// Mitsubishi GX Works2 project: PLC_GROUP7   PLC: FX3G

// global labels: Global1
VAR_GLOBAL
  Switch_Workday AT X007 : BOOL;
  Switch_Cream AT X011 : BOOL;
  Light_Workday AT Y007 : BOOL;
  Light_Transporting0 AT Y000 : BOOL;
  Light_Transporting1 AT Y001 : BOOL;
  Switch_Sample AT X006 : BOOL;
  Light_Chocolate AT Y003 : BOOL;
  Wrap_Krembo AT X000 : BOOL;
  Light_5Krembos AT Y002 : BOOL;
  Stock_Cream AT D1100 : REAL;
  Stock_Chocolate AT D1102 : REAL;
  Stock_Biscuits AT D1104 : REAL;
END_VAR
VAR_GLOBAL CONSTANT
  Serving_Cream : REAL := 300;
  Serving_Chocolate_Normal : REAL := 120;
  Serving_Biscuits : REAL := 6;
  Starting_Cream : REAL := 900;
  Starting_Chocolate : REAL := 500;
  Starting_Biscuits : REAL := 30;
END_VAR
VAR_GLOBAL
  Container_Cream AT D1114 : REAL;
  Container_Chocolate AT D1116 : REAL;
END_VAR
VAR_GLOBAL CONSTANT
  Serving_Chocolate_Double : REAL := 240;
END_VAR
VAR_GLOBAL
  Switch_MachineA AT X010 : BOOL;
  MachineA_on AT M0 : BOOL;
  MachineA_Stop AT X005 : BOOL;
  Sens_30 AT X002 : BOOL;
  Sens_15 AT X001 : BOOL;
  Light_MachineA_Work AT Y004 : BOOL;
  Sens_camera AT X003 : BOOL;
  Light_alternate AT M1 : BOOL;
  Timer_alternate AT TC1 : BOOL;
END_VAR
VAR_GLOBAL CONSTANT
  Timer_alternate_duration : INT := 40;
END_VAR
VAR_GLOBAL
  Timer_alterante_State AT TS1 : BOOL;
  Light_state AT M2 : BOOL;
  Light_Y0_Timer AT TC2 : BOOL;
  Light_Y1_Timer AT TC3 : BOOL;
  Light_Y0_State AT TS2 : BOOL;
  Light_Y1_State AT TS3 : BOOL;
END_VAR
VAR_GLOBAL CONSTANT
  Timer_Alternate_Switch : INT := 5;
END_VAR
VAR_GLOBAL
  Analog_Input1 AT D8280 : INT;
END_VAR
VAR_GLOBAL CONSTANT
  Chocolate_Coat : INT := 5;
  Div_400 : INT := 400;
END_VAR
VAR_GLOBAL
  Dipping_Timer AT TC4 : BOOL;
  Dipping_State AT TS4 : BOOL;
END_VAR
VAR_GLOBAL CONSTANT
  Dipping_Duration : INT := 50;
END_VAR
VAR_GLOBAL
  krembo_dipping AT M3 : BOOL;
END_VAR
VAR_GLOBAL CONSTANT
  krembo_5Limit : INT := 5;
END_VAR
VAR_GLOBAL
  krembo_5Count AT CC1 : BOOL;
  krembo_State AT CS1 : BOOL;
  Counter_5Krembo AT CN1 : INT;
END_VAR
VAR_GLOBAL CONSTANT
  Krembo_6Limit : INT := 6;
END_VAR
VAR_GLOBAL
  Krembo_Second_State AT CS2 : BOOL;
  Counter_6Krembo AT CN2 : INT;
  Krembo_6Count AT CC2 : BOOL;
  Light_Y2_Help AT M5 : BOOL;
  Total_Krembo AT D1118 : REAL;
  Analog_Output AT D8282 : INT;
  Light_Alternate2 AT M4 : BOOL;
  Light_alternate_endDay AT M6 : BOOL;
  Timer_endDay AT TC5 : BOOL;
  Timer_endDay_State AT TS5 : BOOL;
END_VAR
VAR_GLOBAL CONSTANT
  EndDay_Duration : INT := 30;
END_VAR
VAR_GLOBAL
  Light_alternate_endDay2 AT M7 : BOOL;
  Timer_endDay2 AT TC6 : BOOL;
  Timer_endDay_State2 AT TS6 : BOOL;
  Got_Biscuits AT M11 : BOOL;
  Got_Cream AT M12 : BOOL;
  Got_Chocolate AT M13 : BOOL;
  Timer_endDay3 AT TC7 : BOOL;
  Timer_endDay_State3 AT TS7 : BOOL;
  End_Blink_Light2 AT M14 : BOOL;
  Sens_Pack AT X004 : BOOL;
  End_Blink_Light AT M16 : BOOL;
  End_Iteration AT M17 : BOOL;
  Fictive_Light_Workday AT M18 : BOOL;
END_VAR
VAR_GLOBAL CONSTANT
  Mul_40 : INT := 40;
END_VAR

// task Task_01 (event TRUE, interval 0, priority 31): POU_01

PROGRAM POU_01
(* structured ladder/FBD written out as ST: instructions are called as NAME(EN, inputs, outputs); _pN, _eN, _tN stand for wires *)
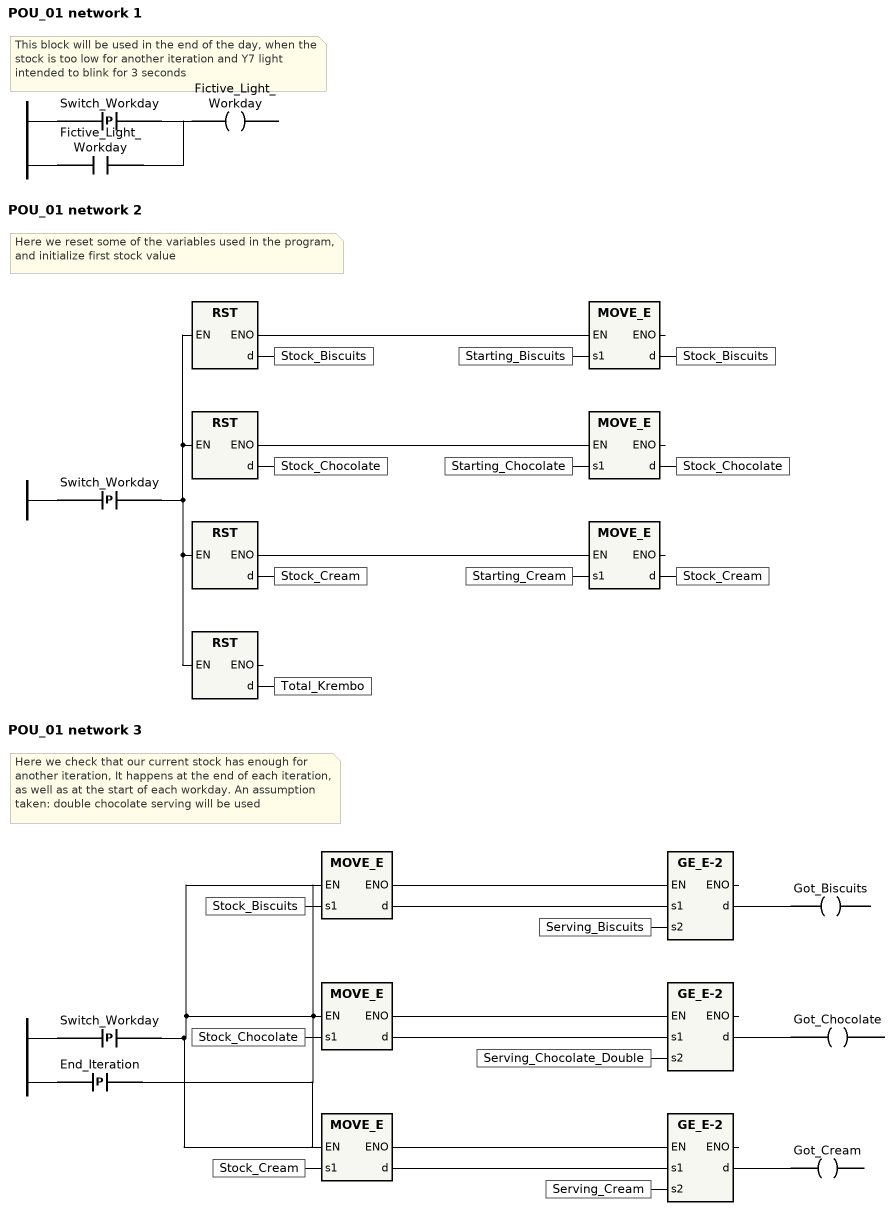
(* network 1 *)
(* This block will be used in the end of the day, when the stock is too low for another iteration and Y7 light intended to blink for 3 seconds *)
Fictive_Light_Workday := LDP(TRUE, Switch_Workday) OR Fictive_Light_Workday;
(* network 2 *)
(* Here we reset some of the variables used in the program, and initialize first stock value *)
_p1 := LDP(TRUE, Switch_Workday);
_e2 := RST(_p1, Stock_Biscuits);
MOVE_E(_e2, Starting_Biscuits, Stock_Biscuits);
_e3 := RST(_p1, Stock_Chocolate);
MOVE_E(_e3, Starting_Chocolate, Stock_Chocolate);
_e4 := RST(_p1, Stock_Cream);
MOVE_E(_e4, Starting_Cream, Stock_Cream);
RST(_p1, Total_Krembo);
(* network 3 *)
(* Here we check that our current stock has enough for another iteration, It happens at the end of each iteration, as well as at the start of each workday. An assumption taken: double chocolate serving will be used *)
_p1 := LDP(TRUE, Switch_Workday) OR LDP(TRUE, End_Iteration);
_e3 := MOVE_E(_p1, Stock_Biscuits, _t2);
GE_E(_e3, _t2, Serving_Biscuits, _t4);
Got_Biscuits := _t4;
_e6 := MOVE_E(_p1, Stock_Chocolate, _t5);
GE_E(_e6, _t5, Serving_Chocolate_Double, _t7);
Got_Chocolate := _t7;
_e9 := MOVE_E(_p1, Stock_Cream, _t8);
GE_E(_e9, _t8, Serving_Cream, _t10);
Got_Cream := _t10;
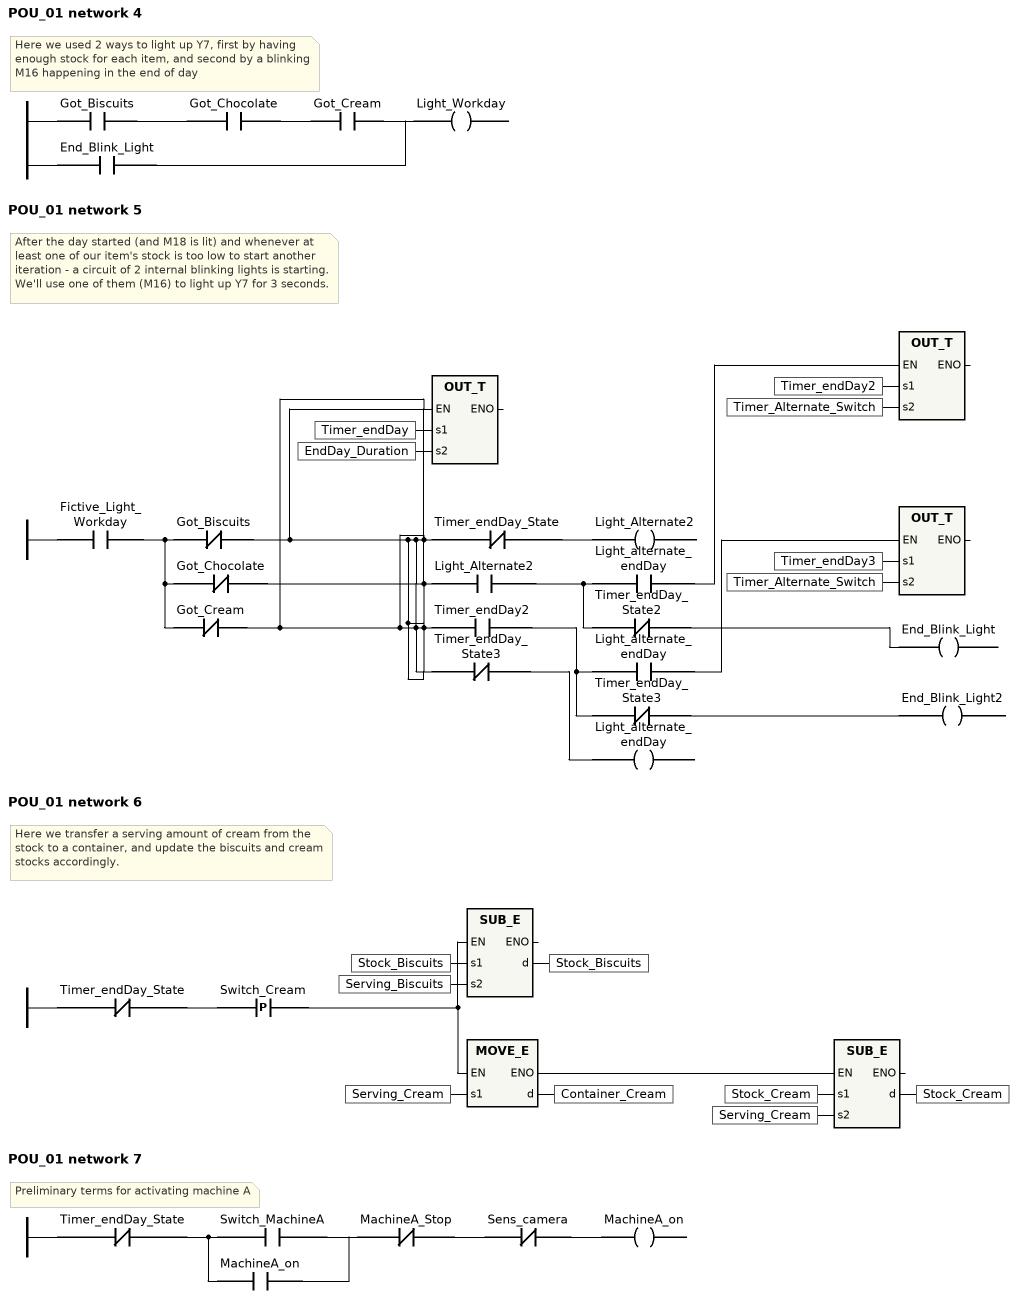
(* network 4 *)
(* Here we used 2 ways to light up Y7, first by having enough stock for each item, and second by a blinking M16 happening in the end of day *)
Light_Workday := (Got_Biscuits AND Got_Chocolate AND Got_Cream) OR End_Blink_Light;
(* network 5 *)
(* After the day started (and M18 is lit) and whenever at least one of our item's stock is too low to start another iteration - a circuit of 2 internal blinking lights is starting. We'll use one of them (M16) to light up Y7 for 3 seconds. *)
_p1 := (Fictive_Light_Workday AND NOT Got_Biscuits) OR (Fictive_Light_Workday AND NOT Got_Chocolate) OR (Fictive_Light_Workday AND NOT Got_Cream);
Light_Alternate2 := _p1 AND NOT Timer_endDay_State;
OUT_T(_p1, Timer_endDay, EndDay_Duration);
_p2 := _p1 AND Light_Alternate2;
OUT_T(_p2 AND Light_alternate_endDay, Timer_endDay2, Timer_Alternate_Switch);
End_Blink_Light := _p2 AND NOT Timer_endDay_State2;
_p3 := _p1 AND Timer_endDay2;
OUT_T(_p3 AND Light_alternate_endDay, Timer_endDay3, Timer_Alternate_Switch);
End_Blink_Light2 := _p3 AND NOT Timer_endDay_State3;
Light_alternate_endDay := _p1 AND NOT Timer_endDay_State3;
(* network 6 *)
(* Here we transfer a serving amount of cream from the stock to a container, and update the biscuits and cream stocks accordingly. *)
_p1 := NOT Timer_endDay_State AND LDP(TRUE, Switch_Cream);
SUB_E(_p1, Stock_Biscuits, Serving_Biscuits, Stock_Biscuits);
_e2 := MOVE_E(_p1, Serving_Cream, Container_Cream);
SUB_E(_e2, Stock_Cream, Serving_Cream, Stock_Cream);
(* network 7 *)
(* Preliminary terms for activating machine A *)
_p1 := NOT Timer_endDay_State;
MachineA_on := (((_p1 AND Switch_MachineA) OR (_p1 AND MachineA_on)) AND NOT MachineA_Stop) AND NOT Sens_camera;
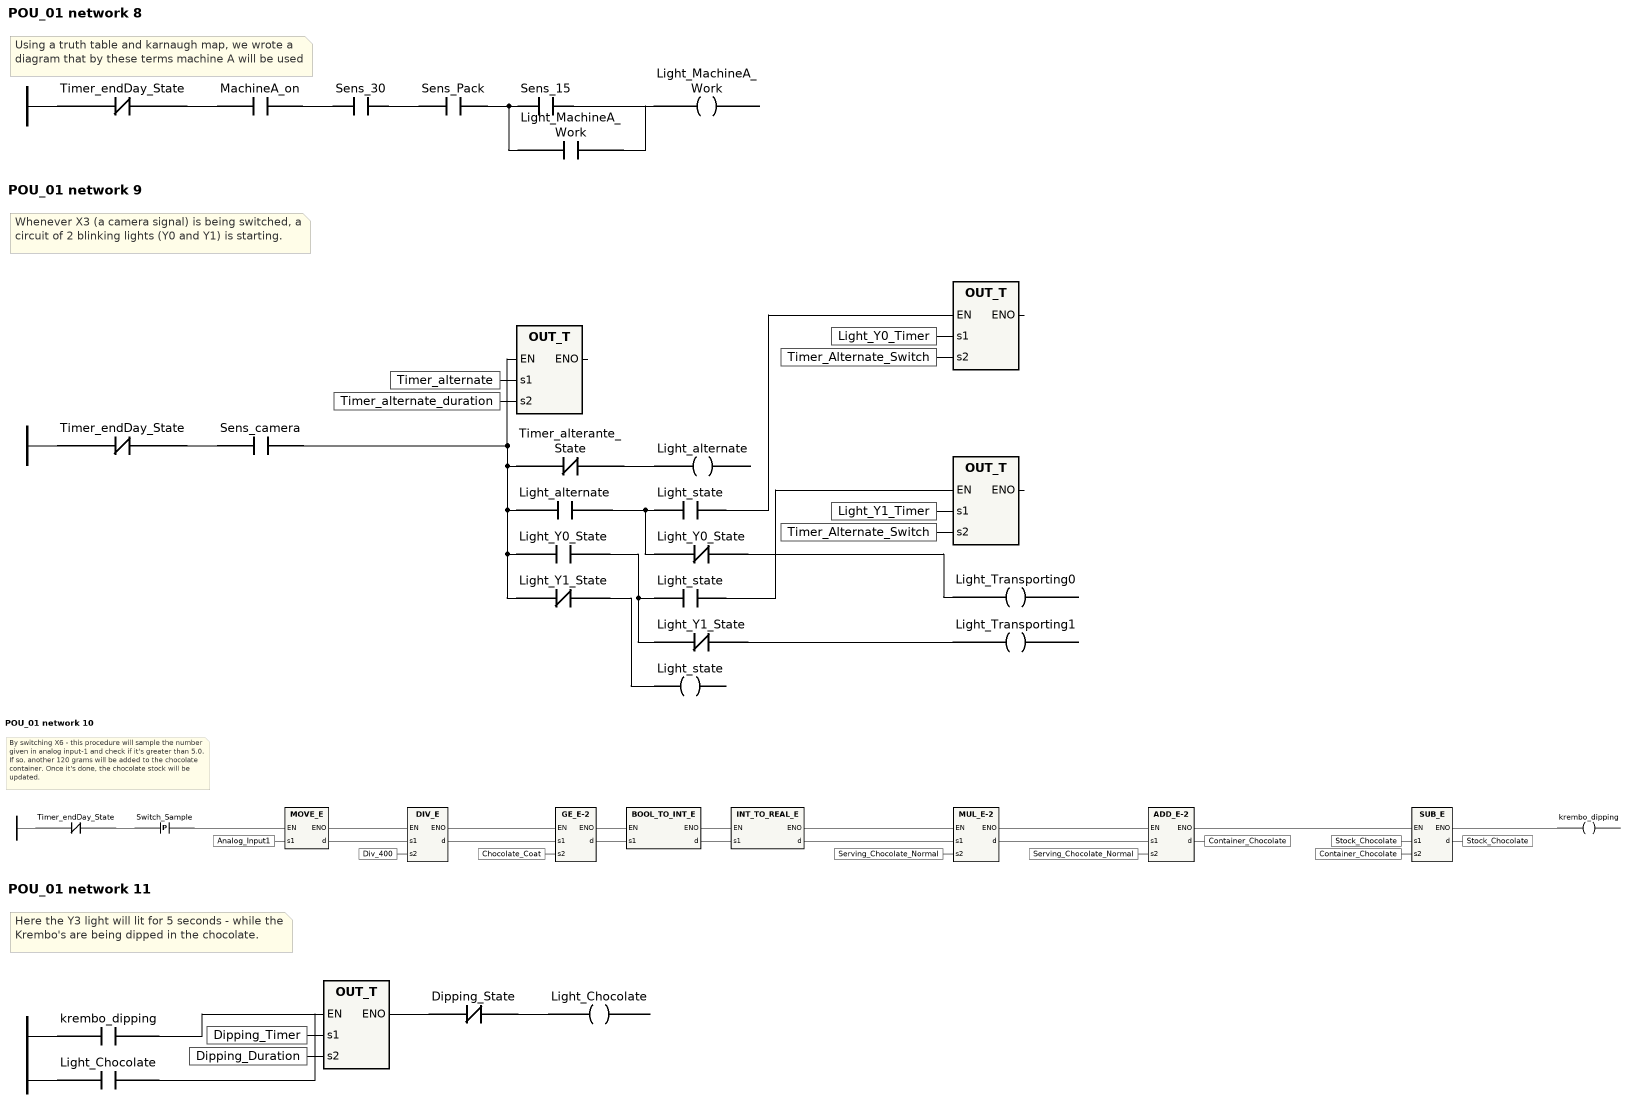
(* network 8 *)
(* Using a truth table and karnaugh map, we wrote a diagram that by these terms machine A will be used *)
_p1 := NOT Timer_endDay_State AND MachineA_on AND Sens_30 AND Sens_Pack;
Light_MachineA_Work := (_p1 AND Sens_15) OR (_p1 AND Light_MachineA_Work);
(* network 9 *)
(* Whenever X3 (a camera signal) is being switched, a circuit of 2 blinking lights (Y0 and Y1) is starting. *)
_p1 := NOT Timer_endDay_State AND Sens_camera;
Light_alternate := _p1 AND NOT Timer_alterante_State;
OUT_T(_p1, Timer_alternate, Timer_alternate_duration);
_p2 := _p1 AND Light_alternate;
OUT_T(_p2 AND Light_state, Light_Y0_Timer, Timer_Alternate_Switch);
Light_Transporting0 := _p2 AND NOT Light_Y0_State;
_p3 := _p1 AND Light_Y0_State;
OUT_T(_p3 AND Light_state, Light_Y1_Timer, Timer_Alternate_Switch);
Light_Transporting1 := _p3 AND NOT Light_Y1_State;
Light_state := _p1 AND NOT Light_Y1_State;
(* network 10 *)
(* By switching X6 - this procedure will sample the number given in analog input-1 and check if it's greater than 5.0. If so, another 120 grams will be added to the chocolate container. Once it's done, the chocolate stock will be updated. *)
_e2 := MOVE_E(NOT Timer_endDay_State AND LDP(TRUE, Switch_Sample), Analog_Input1, _t1);
_e4 := DIV_E(_e2, _t1, Div_400, _t3);
_e6 := GE_E(_e4, _t3, Chocolate_Coat, _t5);
_e8 := BOOL_TO_INT_E(_e6, _t5, _t7);
_e10 := INT_TO_REAL_E(_e8, _t7, _t9);
_e12 := MUL_E(_e10, _t9, Serving_Chocolate_Normal, _t11);
_e13 := ADD_E(_e12, _t11, Serving_Chocolate_Normal, Container_Chocolate);
_e14 := SUB_E(_e13, Stock_Chocolate, Container_Chocolate, Stock_Chocolate);
krembo_dipping := _e14;
(* network 11 *)
(* Here the Y3 light will lit for 5 seconds - while the Krembo's are being dipped in the chocolate. *)
_e1 := OUT_T(krembo_dipping OR Light_Chocolate, Dipping_Timer, Dipping_Duration);
Light_Chocolate := _e1 AND NOT Dipping_State;
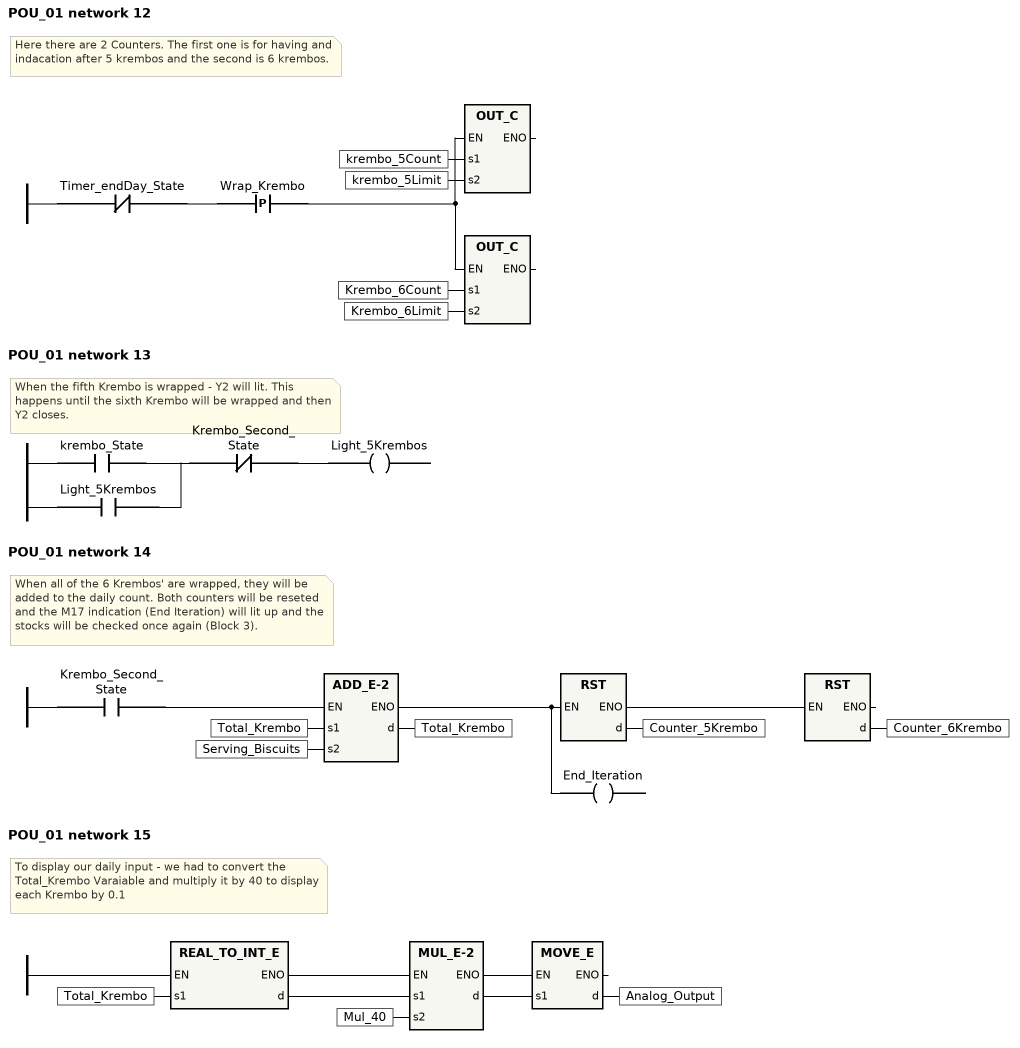
(* network 12 *)
(* Here there are 2 Counters. The first one is for having and indacation after 5 krembos and the second is 6 krembos. *)
_p1 := NOT Timer_endDay_State AND LDP(TRUE, Wrap_Krembo);
OUT_C(_p1, krembo_5Count, krembo_5Limit);
OUT_C(_p1, Krembo_6Count, Krembo_6Limit);
(* network 13 *)
(* When the fifth Krembo is wrapped - Y2 will lit. This happens until the sixth Krembo will be wrapped and then Y2 closes. *)
Light_5Krembos := (krembo_State OR Light_5Krembos) AND NOT Krembo_Second_State;
(* network 14 *)
(* When all of the 6 Krembos' are wrapped, they will be added to the daily count. Both counters will be reseted and the M17 indication (End Iteration) will lit up and the stocks will be checked once again (Block 3). *)
_e1 := ADD_E(Krembo_Second_State, Total_Krembo, Serving_Biscuits, Total_Krembo);
End_Iteration := _e1;
_e2 := RST(_e1, Counter_5Krembo);
RST(_e2, Counter_6Krembo);
(* network 15 *)
(* To display our daily input - we had to convert the Total_Krembo Varaiable and multiply it by 40 to display each Krembo by 0.1 *)
_e2 := REAL_TO_INT_E(TRUE, Total_Krembo, _t1);
_e4 := MUL_E(_e2, _t1, Mul_40, _t3);
MOVE_E(_e4, _t3, Analog_Output);
END_PROGRAM
